{attribute 'qualified_only'}
VAR_GLOBAL
	In : BOOL := 0;
	Out : BOOL := 0;
END_VAR

(* stored: Version 1.1.0.1, ProductVersion 3.1.4024.0
   GVL GVL: Id {5c4e9e9c-f4a4-4375-be14-8edc195f39c3} *)
